(* LS Electric XG5000 project: 23_10_30 *)
(* PLC LSPLC *)

FUNCTION_BLOCK 사칙연산
VAR_INPUT
    IN1 : REAL;
    IN2 : REAL;
END_VAR
VAR_OUTPUT
    ADD_OUT : REAL;
    SUB_OUT : REAL;
    MUL_OUT : REAL;
    DIV_OUT : REAL;
END_VAR

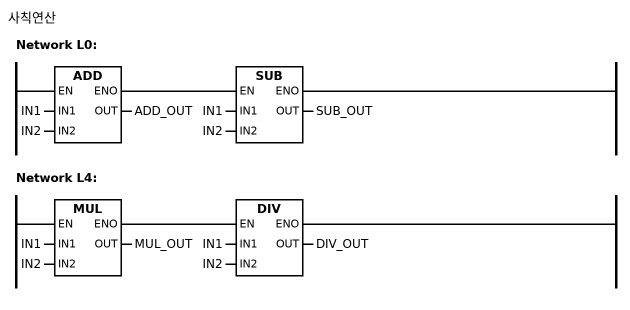
(* Rung L0 *)
ADD_OUT := IN1 + IN2;
SUB_OUT := IN1 - IN2;
(* Rung L4 *)
MUL_OUT := IN1 * IN2;
DIV_OUT := IN1 / IN2;
END_FUNCTION_BLOCK

FUNCTION PITA : REAL
VAR_INPUT
    A변 : REAL;
    B변 : REAL;
END_VAR
VAR
    A제곱 : REAL;
    B제곱 : REAL;
    result : REAL;
    합 : REAL;
END_VAR

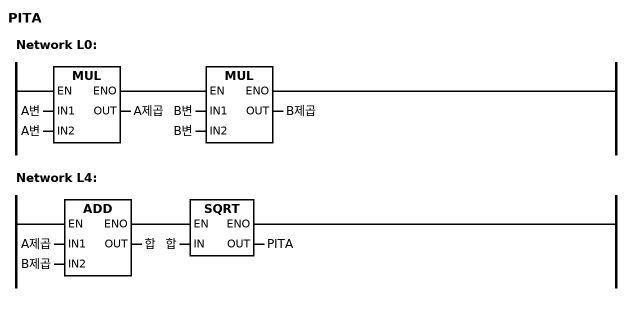
(* Rung L0 *)
A제곱 := A변 * A변;
B제곱 := B변 * B변;
(* Rung L4 *)
합 := A제곱 + B제곱;
PITA := SQRT(합);
END_FUNCTION

FUNCTION_BLOCK 플리커
VAR_INPUT
    FL : BOOL;
    NFL : BOOL;
    OFF : BOOL;
END_VAR
VAR_OUTPUT
    LA1 : BOOL;
    LA2 : BOOL;
END_VAR
VAR
    end : BOOL;
    t1 : TON;
    t2 : TON;
    t3 : TON;
    t4 : TON;
    tp1 : TP;
    tp2 : TP;
    tp3 : TP;
END_VAR

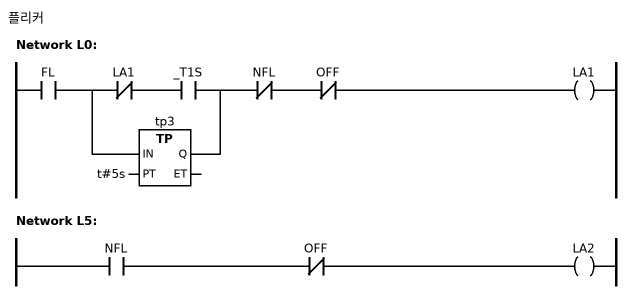
(* Rung L0 *)
tp3(IN := FL, PT := t#5s);
LA1 := ((FL AND NOT LA1 AND _T1S) OR tp3.Q) AND NOT NFL AND NOT OFF;
(* Rung L5 *)
LA2 := NFL AND NOT OFF;
END_FUNCTION_BLOCK

PROGRAM NewProgram (* task: 스캔 프로그램 *)
VAR
    A : REAL := 50.0;
    B : REAL := 8.0;
    CALC : 사칙연산;
    end : BOOL;
    FL : BOOL;
    INST : TON;
    LA1 : BOOL;
    LA2 : BOOL;
    NFL : BOOL;
    OFF : BOOL;
    out : BOOL;
    P1 : BOOL;
    P10 : BOOL;
    P11 : BOOL;
    Q2_P1 : BOOL;
    Q2_P11 : BOOL;
    Q3_P1 : BOOL;
    Q3_P10 : BOOL;
    Q3_P2 : BOOL;
    Q4_P1 : BOOL;
    Q4_P10 : BOOL;
    Q4_P2 : BOOL;
    Q4_P3 : BOOL;
    Q5_P1 : BOOL;
    Q5_P10 : BOOL;
    Q5_P11 : BOOL;
    Q5_P2 : BOOL;
    Q5_P3 : BOOL;
    Q6_OUT : BOOL;
    Q6_P1 : BOOL;
    Q6_P10 : BOOL;
    Q7_P0 : BOOL;
    Q7_P10 : BOOL;
    Q7_T0 : BOOL;
    Q7_t1 : TON;
    Q8_P1 : BOOL;
    Q8_P10 : BOOL;
    Q8_P2 : BOOL;
    Q8_t1 : TON;
    Q8_t2 : TON;
    Q9_P1 : BOOL;
    Q9_P10 : BOOL;
    Q9_T1 : BOOL;
    Q9_ton1 : BOOL;
    result : REAL;
    t1 : TON;
    t2 : TON;
    tp1 : TP;
    tp3 : TP;
    _1 : BOOL;
    플리커 : 플리커;
END_VAR
VAR
    _e1 : R_TRIG;
    _e2 : R_TRIG;
    _e3 : R_TRIG;
    _e4 : R_TRIG;
    _e5 : R_TRIG;
END_VAR

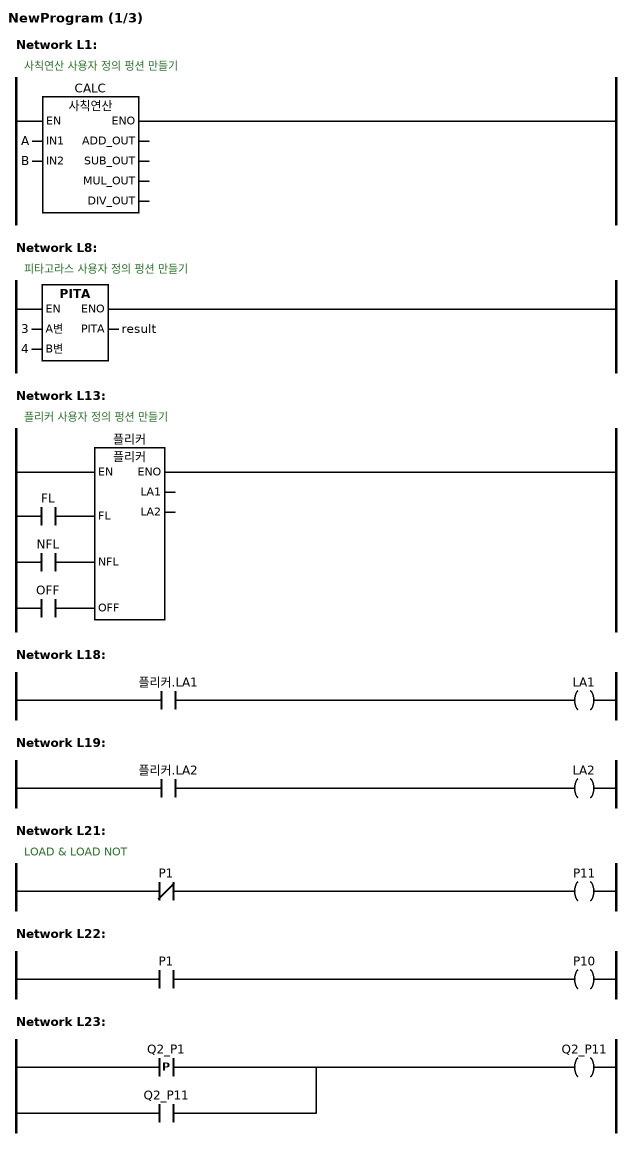
(* 사칙연산 사용자 정의 펑션 만들기 *)
(* Rung L1 *)
CALC(IN1 := A, IN2 := B);
(* 피타고라스 사용자 정의 펑션 만들기 *)
(* Rung L8 *)
result := PITA(A변 := 3, B변 := 4);
(* 플리커 사용자 정의 펑션 만들기 *)
(* Rung L13 *)
플리커(FL := FL, NFL := NFL, OFF := OFF);
(* Rung L18 *)
LA1 := 플리커.LA1;
(* Rung L19 *)
LA2 := 플리커.LA2;
(* LOAD & LOAD NOT *)
(* Rung L21 *)
P11 := NOT P1;
(* Rung L22 *)
P10 := P1;
(* Rung L23 *)
_e1(CLK := Q2_P1);
Q2_P11 := _e1.Q OR Q2_P11;

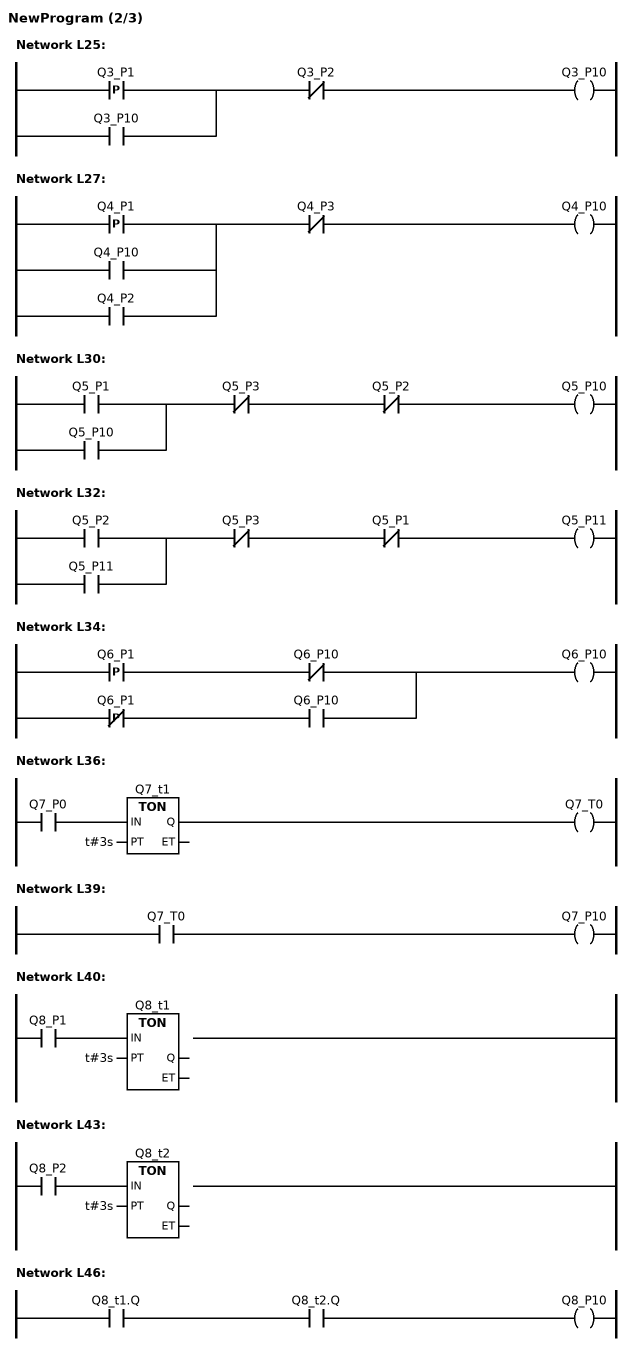
(* Rung L25 *)
_e2(CLK := Q3_P1);
Q3_P10 := (_e2.Q OR Q3_P10) AND NOT Q3_P2;
(* Rung L27 *)
_e3(CLK := Q4_P1);
Q4_P10 := (_e3.Q OR Q4_P10 OR Q4_P2) AND NOT Q4_P3;
(* Rung L30 *)
Q5_P10 := (Q5_P1 OR Q5_P10) AND NOT Q5_P3 AND NOT Q5_P2;
(* Rung L32 *)
Q5_P11 := (Q5_P2 OR Q5_P11) AND NOT Q5_P3 AND NOT Q5_P1;
(* Rung L34 *)
_e4(CLK := Q6_P1);
_e5(CLK := Q6_P1);
Q6_P10 := (_e4.Q AND NOT Q6_P10) OR (NOT _e5.Q AND Q6_P10);
(* Rung L36 *)
Q7_t1(IN := Q7_P0, PT := t#3s);
Q7_T0 := Q7_t1.Q;
(* Rung L39 *)
Q7_P10 := Q7_T0;
(* Rung L40 *)
Q8_t1(IN := Q8_P1, PT := t#3s);
(* Rung L43 *)
Q8_t2(IN := Q8_P2, PT := t#3s);
(* Rung L46 *)
Q8_P10 := Q8_t1.Q AND Q8_t2.Q;

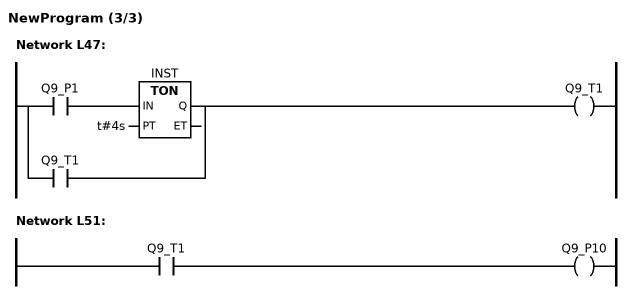
(* Rung L47 *)
INST(IN := Q9_P1, PT := t#4s);
Q9_T1 := INST.Q OR Q9_T1;
(* Rung L51 *)
Q9_P10 := Q9_T1;
END_PROGRAM